{attribute 'no_assign'}
FUNCTION_BLOCK FB_XpMoverState
VAR_INPUT
	eTaskMover 	: E_Movertask;
	refMover	: REFERENCE TO MC_PlanarMover;
	bResetMover	: BOOL;
END_VAR
VAR_OUTPUT
	bDoneMover 		:BOOL;
END_VAR
VAR
	MSFeedback			: ARRAY [0..30] OF MC_PlanarFeedback;
	
//	bDoneMover			: BOOL;
	nMoverState			: INT;
	//eTaskMover			: E_MOVERTASK;
	
	stOption			: ST_MoveOnTrackOptions;
	Constraint			: DynamicConstraint_PathXY;
	Constraint_c		: DynamicConstraint_Coordinates;
	stoption_c			: ST_MoveCOptions;
	stOption_j			: ST_JoinTrackOptions;
	i: INT;
	ValueC : LREAL := 300;
END_VAR

(*
IF NOT __ISVALIDREF(refMover) THEN
	RETURN;
END_IF
*)

IF bResetMover THEN
	bResetMover := FALSE;
	nMoverState := 0;
	RETURN;
END_IF

CASE nMoverState OF
	0://IDLE
	IF eTaskMover =E_MoverTask.IDLE THEN //IDLE状態で0に戻ったらbDoneMoverを0に戻す
	bDoneMover := FALSE;
	END_IF
	
		CASE eTaskMover OF
			E_MoverTask.JOIN_T2 		: nMoverState :=100;
			E_MoverTask.JOIN_T3			: nMoverState :=200;
			E_MoverTask.MOVE_END_T1		: nMoverState :=300;
			E_MoverTask.MOVE_HALF_T2	: nMoverState :=400;
			E_MoverTask.MOVE_TO_T2 		: nMoverState :=500;
			E_MoverTask.MOVE_TO_T3 		: nMoverState :=600;
			E_MoverTask.MOVE_BEHIND_T1	: nMoverState :=700;
			E_Movertask.RESET_ERROR		: nMoverState :=950;
		END_CASE
	
	
	100://JOIN T2
	refMover.JoinTrack(commandFeedback:= MSFeedback[0], 
				targetTrack:= GVL.XpTrack[2], 
				constraint:= constraint, 
				options:= stOption_j);
	nMoverState:=101;
	
	101:
	IF (MSFeedback[0].Active OR MSFeedback[0].Done) THEN
		nMoverState:=102;
	END_IF	
	
	102:
	IF MSFeedback[0].Done THEN
		bDoneMover := TRUE;
		nMoverState := 0;
	END_IF


	200://JOIN T3
	refMover.JoinTrack(commandFeedback:= MSFeedback[1], 
				targetTrack:= GVL.XpTrack[3], 
				constraint:= constraint, 
				options:= stOption_j);
	nMoverState:=201;
	
	201:
	IF (MSFeedback[1].Active OR MSFeedback[1].Done) THEN
		nMoverState:=202;
	END_IF	
	
	202:
	IF MSFeedback[1].Done THEN
		bDoneMover := TRUE;
		nMoverState := 0;
	END_IF
	
	
	300://MOVE T1
	refMover.MoveOnTrack(
		commandFeedback:= MSFeedback[2], 
		targetTrack:= GVL.XpTrack[1], 
		targetPositionOnTrack:= GVL.Xptrack[1].GetLength(), 
		constraint:= Constraint, 
		options:= stOption);
		nMoverState:=301;
		
	301:
	IF (MSFeedback[2].Active OR MSFeedback[2].Done) THEN
		nMoverState:=302;
	END_IF	
	
	302:
	IF MSFeedback[2].Done THEN
		bDoneMover := TRUE;
		nMoverState := 0;
	END_IF
	
	
	400://MOVE T2 HALF
	refMover.MoveOnTrack(
		commandFeedback:= MSFeedback[3], 
		targetTrack:= GVL.XpTrack[2], 
		targetPositionOnTrack:= GVL.XpTrack[2].GetLength()/2, 
		constraint:= Constraint, 
		options:= stOption);
		nMoverState:=401;
		
	401:
	IF (MSFeedback[3].Active OR MSFeedback[3].Done) THEN
		nMoverState:=402;
	END_IF	
	
	402:
	IF MSFeedback[3].Done THEN
		bDoneMover := TRUE;
		nMoverState := 0;
	END_IF	
	
	
	500://MOVE T2 END
	refMover.MoveOnTrack(
		commandFeedback:= MSFeedback[4], 
		targetTrack:= GVL.XpTrack[2], 
		targetPositionOnTrack:= GVL.Xptrack[2].GetLength(), 
		constraint:= Constraint, 
		options:= stOption);
			nMoverState:=501;
		
	501:
	IF (MSFeedback[4].Active OR MSFeedback[4].Done) THEN
		nMoverState:=502;
	END_IF	
	
	502:
	IF MSFeedback[4].Done THEN
		bDoneMover := TRUE;
		nMoverState := 0;
	END_IF	
	
	600://MOVE T3
	refMover.MoveOnTrack(
		commandFeedback:= MSFeedback[5], 
		targetTrack:= GVL.XpTrack[3], 
		targetPositionOnTrack:= GVL.XpTrack[3].GetLength(), 
		constraint:= Constraint, 
		options:= stOption);
		nMoverState:=601;
		
	601:
	IF MSFeedback[5].Active OR MSFeedback[5].Done THEN
		nMoverState:=602;
	END_IF	
	
	602:
	IF MSFeedback[5].Done THEN
		bDoneMover := TRUE;
		nMoverState := 0;
	END_IF	
	
	700://MOVE BIHIND T1
		refMover.MoveOnTrack(
		commandFeedback:= MSFeedback[6], 
		targetTrack:= GVL.XpTrack[1], 
		targetPositionOnTrack:= GVL.Xptrack[1].GetLength()/2, 
		constraint:= Constraint, 
		options:= stOption);
		nMoverState:=701;
		
	701:
	IF (MSFeedback[6].Active OR MSFeedback[6].Done) THEN
		nMoverState:=702;
	END_IF	
	
	702:
	IF MSFeedback[6].Done THEN
		bDoneMover := TRUE;
		nMoverState := 0;
	END_IF	
	
	950:
	refMover.Reset(commandFeedBack :=MSFeedback[30]);
	nMoverState :=951;
	
	951:
	IF MSFeedback[30].Active OR MSFeedback[30].Done THEN
		nMoverState :=952;
	END_IF
	
	952:
	IF MSFeedback[30].Done THEN
		bDoneMover :=TRUE;
		nMoverState := 0;
	END_IF
		
END_CASE

Constraint.SetValuesVADJ(
		V:= 100, 
		A:= 7000, 
		D:= 7000,
		J:=35000);
		
Constraint_c.SetLimit(
	Coordinate:= Coord_Mcs_C1, 
	V:= ValueC, 
	A:= 7000, 
	D:= 7000, 
	J:= 35000);

(*
refMover.Update();
*)
FOR i:=0 TO 30 DO
	MSFeedback[i].Update();
END_FOR

END_FUNCTION_BLOCK

(* stored: Version 1.1.0.1
   POU FB_XpMoverState: Id {a226981c-08b8-49d9-b98e-32c36b71e77d}, SpecialFunc None *)
